(*Implements MoveRequest interface for EPICS Motor*)
FUNCTION_BLOCK FB_EpicsMoveRequest IMPLEMENTS I_MoveRequest
VAR
   // EPICS Interface
    {attribute 'no_copy'}
    stMotionCommand : REFERENCE TO ST_MotionCommand;
	{attribute 'no_copy'}
	stMotionStatus:  REFERENCE TO ST_MotionStatus;
	
    eEnableMode: E_StageEnableMode:=E_StageEnableMode.DURING_MOTION;
    bMoveCmd	: BOOL;
    {attribute 'hide'}
    eHomeMode	: E_EpicsHomeCmd := E_EpicsHomeCmd.NONE;
    {attribute 'hide'}
    bEnableDone : BOOL;
    {attribute 'hide'}
    bMoveOk: BOOL;
    (* non epics*)
    {attribute 'hide'}
    bExecute : BOOL;
    {attribute 'hide'}
    rtMoveCmdShortcut: R_TRIG;
    {attribute 'hide'}
    rtHomeCmdShortcut: R_TRIG;
    {attribute 'hide'}
    rtEnableMode: R_TRIG;
    {attribute 'hide'}
    rtNewMoveReq: R_TRIG;
    {attribute 'hide'}
    rtUserExec: R_TRIG;
    {attribute 'hide'}
    rtExec : R_TRIG;
    {attribute 'hide'}
    stMotionRequestStatus : ST_MoveRequestStatus;
    {attribute 'hide'}
    ftStopExec: F_TRIG;
    {attribute 'hide'}
    eRestoreSettingsState : ( RestoreSettingWaiting:=0, RestoreSettingDone:=1);
    {attribute 'hide'}
    ftstop: F_TRIG;
	rtExecute : R_TRIG;
END_VAR

IF NOT __ISVALIDREF( stMotionCommand ) OR NOT  __ISVALIDREF( stMotionStatus ) THEN
   RETURN;
END_IF
(* Check for the plc shortcut commands
   Used for testing or to circumvent motor record issues*)
rtMoveCmdShortcut(CLK:=bMoveCmd);
rtHomeCmdShortcut(CLK:=stMotionCommand.bHomeCmd);

(* Execute on rising edge*)
IF rtMoveCmdShortcut.Q AND NOT stMotionCommand.bExecute THEN
    stMotionCommand.bExecute:=TRUE;
    stMotionCommand.nCommand := E_EpicsMotorCmd.MOVE_ABSOLUTE;

ELSIF rtHomeCmdShortcut.Q AND NOT stMotionCommand.bExecute THEN

    IF (*( eHomeMode = E_EpicsHomeCmd.ABSOLUTE_SET )  OR*) ( eHomeMode = E_EpicsHomeCmd.NONE) THEN
       stMotionCommand.bExecute:= FALSE;
    ELSE
       stMotionCommand.bExecute:= TRUE;
    END_IF
    stMotionCommand.nCommand:=E_EpicsMotorCmd.HOME;
    (* Automatically fill the correct nCmdData for homing*)
    stMotionCommand.nCmdData:=eHomeMode;
END_IF

(* entry point for local and EPICS main execs *)
rtUserExec(CLK:=stMotionCommand.bExecute);
(* if a Move/Home Goal is comfirmed and there is no persistant
   error conditions, then we have a valid move request.*)
stMotionRequestStatus.bNewMoveReq S= NOT stMotionStatus.bBusy AND rtUserExec.Q AND NOT stMotionStatus.bError AND bMoveOk;;
(* this Move request is valid till an error occurs or the currently move is done *)
stMotionRequestStatus.bNewMoveReq R= NOT stMotionCommand.bExecute OR stMotionStatus.bError;
stMotionRequestStatus.bPrepareDisable R= stMotionRequestStatus.bNewMoveReq;
rtNewMoveReq(CLK:=stMotionRequestStatus.bNewMoveReq);

(* Set the proper command for the request move;
   if bservo not set, manual step moves will be performed *)
IF rtUserExec.Q THEN
    // Transfer nCommand and nCmdData to local copies at rising edge of bExecute (avoid issues if nCommand or nCmdData are changed during a command)
    stMotionRequestStatus.nCmdData:=stMotionCommand.nCmdData;
    stMotionRequestStatus.nCommand:=stMotionCommand.nCommand;
    IF NOT stMotionCommand.bHomeCmd THEN
        (* attempting to move an axis without homing first? *)
        IF eHomeMode <> E_EpicsHomeCmd.NONE AND NOT stMotionStatus.bHomed THEN
            (* one can just set bHome here even though no homing was done?*)
            stMotionStatus.sErrorMessage:='Axis homing mode set, but homing routine pending';
        END_IF
    END_IF
END_IF

rtEnableMode(CLK:=(eEnableMode = E_StageEnableMode.DURING_MOTION));
(* Handle auto-enable timing *)
CASE eEnableMode OF
    (* Not recommended, not tested *)
    E_StageEnableMode.ALWAYS:
        // if no latching interlock condition, No errors
        stMotionRequestStatus.bEnable:= NOT stMotionStatus.bError AND bMoveOk;
    E_StageEnableMode.DURING_MOTION:
        IF rtEnableMode.Q THEN
            stMotionRequestStatus.bEnable := FALSE;
        END_IF
        IF rtNewMoveReq.Q THEN
            stMotionRequestStatus.bEnable S= stMotionRequestStatus.bNewMoveReq;
        END_IF
END_CASE

stMotionRequestStatus.bExecute := NOT stMotionStatus.bError AND stMotionCommand.bExecute AND bEnableDone;
stMotionRequestStatus.bExecHome:=stMotionRequestStatus.bExecute AND stMotionRequestStatus.nCommand = 10;
stMotionRequestStatus.bExecMove:=stMotionRequestStatus.bExecute AND NOT stMotionRequestStatus.bExecHome;

// Declare axis busy earlier and clear previous done state
rtExecute(CLK:=stMotionCommand.bExecute);
IF rtExecute.Q THEN
	InitMoveRequest();
END_IF

// release epics and local interface
bMoveCmd := FALSE;
stMotionCommand.bHomeCmd := FALSE;

// Move done, or aborted? prepare disable.
// we'll wait for axis to be in standstill and this state machine to be idling.
ftStopExec(CLK:=stMotionCommand.bExecute);
stMotionRequestStatus.bPrepareDisable S= (eEnableMode=E_StageEnableMode.DURING_MOTION) AND ftStopExec.Q;

IF stMotionStatus.bBusy THEN
    stMotionStatus.sErrorMessage := '';
END_IF

//ftstop(CLK:=stMotionInterface.bExecute);

METHOD PUBLIC CallAfterInit
VAR_INPUT
    stMotionCommand : REFERENCE TO ST_MotionCommand;
	stMotionStatus:  REFERENCE TO ST_MotionStatus;
END_VAR
THIS^.stMotionCommand REF=stMotionCommand;
THIS^.stMotionStatus REF=stMotionStatus;
END_METHOD

METHOD ClearMoveRequest
// falling edge here when target is reached, move halted
stMotionCommand.bExecute := FALSE;
stMotionStatus.bDone := FALSE;
stMotionStatus.bBusy := FALSE;
// release the cmds
stMotionCommand.bHomeCmd:=FALSE;
bMoveCmd:=FALSE;
END_METHOD

METHOD ClearMoveRequestErrors
stMotionStatus.bError := FALSE;
stMotionStatus.nErrorId := 0;
stMotionStatus.sErrorMessage := '';
stMotionRequestStatus.bExecute := FALSE;
END_METHOD

PROPERTY EnableMode : ENUM_StageEnableMode
GET
EnableMode := eEnableMode;
END_GET
SET
eEnableMode := EnableMode;
END_SET
END_PROPERTY

//FB_Init is always available implicitly and it is used primarily for initialization.
//The return value is not evaluated. For a specific influence, you can also declare the
//methods explicitly and provide additional code there with the standard initialization
//code. You can evaluate the return value.
METHOD FB_Init: BOOL
VAR_INPUT
    bInitRetains: BOOL; // TRUE: the retain variables are initialized (reset warm / reset cold)
    bInCopyCode: BOOL;  // TRUE: the instance will be copied to the copy code afterward (online change)
    stMotionCommand : REFERENCE TO ST_MotionCommand;
	stMotionStatus:  REFERENCE TO ST_MotionStatus;
END_VAR
THIS^.stMotionCommand REF=stMotionCommand;
THIS^.stMotionStatus REF=stMotionStatus;
END_METHOD

METHOD HaltMoveRequest : BOOL
VAR_INPUT
    Busy	: BOOL;
END_VAR
// Halt is always a user stop but not an interlock event or a reset.
HaltMoveRequest := NOT stMotionCommand.bReset AND ftstop.Q
                        AND ((Busy AND (stMotionRequestStatus.nCommand=10))
                        OR (Busy AND (stMotionRequestStatus.nCommand=3)));
END_METHOD

PROPERTY INTERNAL HomeCmd : BOOL
SET
stMotionCommand.bHomeCmd := HomeCmd;
END_SET
END_PROPERTY

{attribute 'monitoring' := 'variable'}
PROPERTY INTERNAL HomeMode : E_EpicsHomeCmd
SET
eHomeMode := HomeMode;
END_SET
END_PROPERTY

METHOD InitMoveRequest
stMotionStatus.bBusy := TRUE;
stMotionStatus.bDone := FALSE;
// reset error flag
stMotionStatus.sErrorMessage := '';
END_METHOD

PROPERTY INTERNAL MoveCmd : BOOL
SET
bMoveCmd := MoveCmd;
END_SET
END_PROPERTY

METHOD MoveRequest
VAR_INPUT
    // From Axis through the drive
    EnableDone	: BOOL;
    // From Interlock through the drive
    MoveOk  : BOOL;
END_VAR
THIS^.bMoveOk := MoveOk;
THIS^.bEnableDone := EnableDone;
END_METHOD

(*Internal use only purpose*)
METHOD INTERNAL MoveRequestCmds
VAR_INPUT
    (* From Drive*)
    HomeCmd	: BOOL;
    MoveCmd	: BOOL;
    HomeMode	: E_EpicsHomeCmd := E_EpicsHomeCmd.NONE;
    EnableMode	: E_StageEnableMode :=  E_StageEnableMode.DURING_MOTION;
END_VAR
THIS^.stMotionCommand.bHomeCmd := HomeCmd;
THIS^.eHomeMode := HomeMode;
THIS^.eEnableMode := EnableMode;
THIS^.bMoveCmd	:= MoveCmd;
END_METHOD

METHOD MoveRequestCompleted
VAR_INPUT
    MoveDone : BOOL;
    HomeDone : BOOL;
END_VAR
stMotionStatus.bHomed := HomeDone;
ClearMoveRequest();
MoveRequestDone(Done:=MoveDone OR HomeDone);
END_METHOD

METHOD MoveRequestDone
VAR_INPUT
    Done : BOOL;
END_VAR
stMotionStatus.bDone := Done;
END_METHOD

METHOD MoveRequestError
VAR_INPUT
    Error :BOOL;
    ErrorId :UDINT;
    ErrorMessage:T_MAXSTRING;
END_VAR
stMotionStatus.bError := Error;
stMotionStatus.nErrorId := ErrorId;
stMotionStatus.sErrorMessage:= ErrorMessage;

IF Error THEN
	ClearMoveRequest();
END_IF
END_METHOD

METHOD MoveResetDone
THIS^.stMotionCommand.bReset := FALSE;
END_METHOD

METHOD ResetMoveEnable
IF stMotionRequestStatus.bPrepareDisable THEN
    IF THIS^.eEnableMode=E_StageEnableMode.DURING_MOTION THEN
        THIS^.stMotionRequestStatus.bEnable := FALSE;
    END_IF
    THIS^.stMotionRequestStatus.bPrepareDisable := FALSE;
END_IF
END_METHOD

METHOD ResetMoveRequest
END_METHOD

METHOD RestoreSettings
VAR_INPUT
    RestoreDone : BOOL;
    SavedPosition : LREAL;
END_VAR
// no needed in production since the actual position is already set on the axis
// and epics status will get that last position
// use this to restore anything thats not an axisref paramter.

CASE eRestoreSettingsState OF
    RestoreSettingWaiting:
        IF RestoreDone THEN
            THIS^.stMotionCommand.fPosition := SavedPosition;
            eRestoreSettingsState := RestoreSettingDone;
        END_IF
    RestoreSettingDone:;

END_CASE
END_METHOD

PROPERTY INTERNAL RestoreSettingsState : UINT
GET
//RestoreSettingsState := eRestoreSettingsState;
END_GET
END_PROPERTY

PROPERTY Status : REFERENCE TO ST_MoveRequestStatus
GET
Status REF= stMotionRequestStatus;
END_GET
END_PROPERTY

END_FUNCTION_BLOCK

(* stored: Version 1.1.0.1
   POU FB_EpicsMoveRequest: Id {f9713c0b-09a1-45a0-9fc6-342a7422cfa5}, SpecialFunc None
   Method CallAfterInit: Id {c5f4a41a-2a36-4ec0-b020-e8f39761af26}
   Method ClearMoveRequest: Id {fc3a5981-a4d7-4a2d-bb30-c09c583c9e55}
   Method ClearMoveRequestErrors: Id {2bb41509-e70c-4465-a06c-a29812268b06}
   Property EnableMode: Id {9356bd40-5ede-4c8b-b065-3ca414d58ac7}
   Get Get: Id {0f06a9c5-786f-4b36-9ffb-1932b02bcacd}
   Set Set: Id {21b092e9-96af-46ee-9d8d-c77dcd117d11}
   Method FB_Init: Id {9133e91c-1e17-4b3b-aa68-c9be539e6510}
   Method HaltMoveRequest: Id {71c9e391-cb0d-4362-ab43-3cfd1f6c0962}
   Property HomeCmd: Id {0f71e1ab-8145-4742-9a26-f8968cdf5f7f}
   Set Set: Id {62647b23-69df-401c-9527-d1a9db32685c}
   Property HomeMode: Id {e2310f41-6785-4f5a-8351-c40e1e907fe6}
   Set Set: Id {398bedac-ab14-4d81-8298-42677f728951}
   Method InitMoveRequest: Id {2d590fc6-f95b-45d5-9e1d-141474a0f09b}
   Property MoveCmd: Id {00f2db26-21fd-456b-8b0d-f7ac8b74db84}
   Set Set: Id {7f2e6fc9-61d1-4f81-b80f-6806642b691d}
   Method MoveRequest: Id {664b6655-0949-47c1-b45f-a64c7d0cda3b}
   Method MoveRequestCmds: Id {d84ff316-c87c-445b-b337-4ae6bc661e04}
   Method MoveRequestCompleted: Id {29932e68-9af9-4521-bd55-b747e571b46c}
   Method MoveRequestDone: Id {ab10537f-2bb4-4a28-9c3a-e3028ea8d9fc}
   Method MoveRequestError: Id {674719eb-75b4-4cc3-924b-ecc3d1af31ff}
   Method MoveResetDone: Id {f2401880-c9b3-4971-9d2e-b338ef5fea0a}
   Method ResetMoveEnable: Id {f28760d0-5752-4bf4-b850-362b1de6a659}
   Method ResetMoveRequest: Id {90fe06b0-aa4b-458a-9f0e-28628dab07b6}
   Method RestoreSettings: Id {08281416-55cb-4b9c-81b3-3cf6fd0d7faf}
   Property RestoreSettingsState: Id {b366cb5d-502b-43b3-8623-320516670b00}
   Get Get: Id {a39741db-d8b0-422d-b3ab-4a4dba01333b}
   Property Status: Id {f678d159-cc5d-41ad-889c-5f951c755b6f}
   Get Get: Id {08876ea6-b526-4166-bd4c-0a2aa1b11215} *)
